(*			
	RafalOS
	Rafał Osajda		20.11.2025		TC 4024.66
	Interfejs przekazywany do modułów tworzących strony
*)
INTERFACE ITF_MCHMIMachineControl_HMI_PrepScr_06_XX

METHOD PUBLIC GetActiveModeName : ST_BaseLabel
VAR_INPUT
END_VAR
END_METHOD

METHOD PUBLIC GetActiveStateName : ST_BaseLabel
VAR_INPUT
END_VAR
END_METHOD

END_INTERFACE

(* stored: Version 1.1.0.1
   Itf ITF_MCHMIMachineControl_HMI_PrepScr_06_XX: Id {efea9608-1c25-0161-24f5-512510b46507}
   Method GetActiveModeName: Id {239c7565-46be-07aa-3fbc-99dcca9c8ba1}
   Method GetActiveStateName: Id {03ad543d-2706-0245-3071-13f8b151d31f} *)
